TYPE ST_IO2_DoubleInputLockedCtrl :
STRUCT
	eInputSource			: E_IO2_InputSource;
	sInputName		: STRING(40);

	eTypeInput1			: E_IO2_Type;
	tTimeOnFilter1			: TIME;
	tTimeOffFilter1			: TIME;
	tTimeLatch1			: TIME;

	eTypeInput2			: E_IO2_Type;
	tTimeOnFilter2			: TIME;
	tTimeOffFilter2			: TIME;
	tTimeLatch2			: TIME;
END_STRUCT
END_TYPE

(* stored: Version 1.1.0.1, ProductVersion 3.1.4024.15
   DUT ST_IO2_DoubleInputLockedCtrl: Id {54a6833a-b2cf-4566-a7c3-e936f34d08a2} *)
